FUNCTION_BLOCK SWITCH (* Switch(demultiplex)an event *)
  (* Standard: 61499-1; Classification: Event Processing; Function: Event Switch *)
  (* Version 7.0, 01/12/2011, LAPAS, UDESC *)
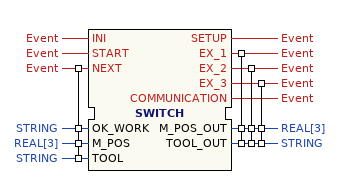
  EVENT_INPUT
    INI; (* Inicializa o bloco *)
    START; (* Inicia o primeiro evento de saida *)
    NEXT WITH OK_WORK, M_POS, TOOL; (* Gera o proximo evento de saida *)
  END_EVENT
  EVENT_OUTPUT
    SETUP; (* Setup da maquina *)
    EX_1 WITH M_POS_OUT, TOOL_OUT; (* Executable 1 *)
    EX_2 WITH M_POS_OUT, TOOL_OUT; (* Executable 2 *)
    EX_3 WITH M_POS_OUT, TOOL_OUT; (* Executable 3 *)
    COMMUNICATION; (* comunicacao *)
  END_EVENT
  VAR_INPUT
    OK_WORK : STRING;
    M_POS : ARRAY [0..2] OF REAL;
    TOOL : STRING;
  END_VAR
  VAR_OUTPUT
    M_POS_OUT : ARRAY [0..2] OF REAL;
    TOOL_OUT : STRING;
  END_VAR
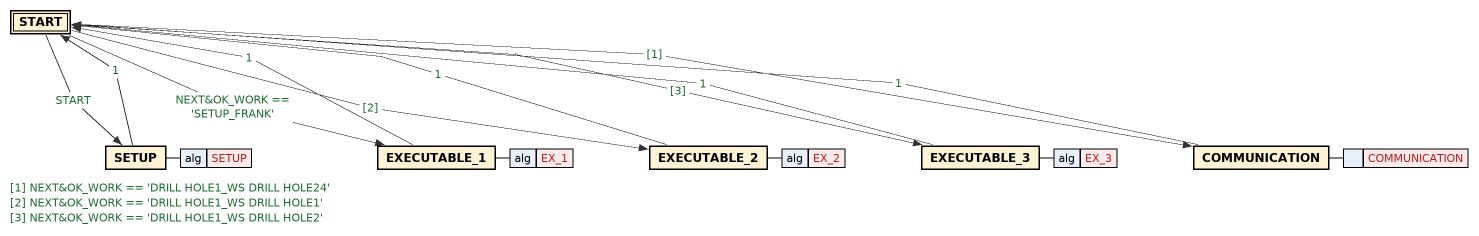
  EC_STATES
    START;
    SETUP : alg -> SETUP;
    EXECUTABLE_1 : alg -> EX_1;
    EXECUTABLE_2 : alg -> EX_2;
    EXECUTABLE_3 : alg -> EX_3;
    COMMUNICATION : -> COMMUNICATION;
  END_STATES
  EC_TRANSITIONS
    START TO SETUP := START;
    START TO EXECUTABLE_1 := NEXT&OK_WORK == 'SETUP_FRANK';
    START TO EXECUTABLE_2 := NEXT&OK_WORK == 'DRILL HOLE1_WS DRILL HOLE1';
    START TO EXECUTABLE_3 := NEXT&OK_WORK == 'DRILL HOLE1_WS DRILL HOLE2';
    START TO COMMUNICATION := NEXT&OK_WORK == 'DRILL HOLE1_WS DRILL HOLE24';
    SETUP TO START := 1;
    EXECUTABLE_1 TO START := 1;
    EXECUTABLE_2 TO START := 1;
    EXECUTABLE_3 TO START := 1;
    COMMUNICATION TO START := 1;
  END_TRANSITIONS
END_FUNCTION_BLOCK
(* other elements stored in the file *)
(* Algorithm Name=alg *)
(* Lua Text=M_POS_OUT[1] = M_POS[1] M_POS_OUT[2] = M_POS[2] M_POS_OUT[3] = M_POS[3] *)
